// TIA Portal V19 program export: 2 tag tables, 0 data types, 0 data blocks, 1 code blocks (in call order from the OBs), 0 instance data blocks

VAR_GLOBAL   // PLC tag table "Default tag table"
   memstart1 AT %M2.2 : Bool;
END_VAR

VAR_GLOBAL   // PLC tag table "driver"
   "Start Button 0" AT %I0.0 : Bool;
   "Stop Button 0" AT %I0.1 : Bool;
   "Selector 0 (State 0)" AT %I0.2 : Bool;
   "jog left" AT %I0.3 : Bool;
   "jog right" AT %I0.4 : Bool;
   "Potentiometer 0 (V)" AT %IW100 : Int;
   "Belt Conveyor (6m) 0 (V)" AT %QW100 : Int;
   "mem-edge1" AT %M0.0 : Bool;
   "mem-edge2" AT %M0.1 : Bool;
   "mem-edge3" AT %M0.2 : Bool;
   "mem-edge4" AT %M0.3 : Bool;
   "mem-edge5" AT %M0.4 : Bool;
   "memory-start" AT %M1.0 : Bool;
   "memory-stop" AT %M1.1 : Bool;
   "memory-3" AT %M1.2 : Bool;
   "memory-4" AT %M1.3 : Bool;
   "memory-5" AT %M1.4 : Bool;
   "mem-out scale" AT %MD100 : Real;
   "mem-val" AT %MW20 : Int;
   "mem-out norm" AT %MD104 : Real;
   "mem-jog-left" AT %MD108 : Real;
   "mem-jog-right" AT %MD112 : Real;
   spead AT %MD116 : Real;
   spead_enter AT %MD120 : Real;
END_VAR

ORGANIZATION_BLOCK "Main"   // OB1, LAD, ProgramCycle
TITLE = "Main Program Sweep (Cycle)"
{ S7_Optimized_Access := 'TRUE' }
// stored: SetENOAutomatically false
   VAR_INPUT
      Initial_Call : Bool;   // Initial call of this OB
      Remanence : Bool;   // =True, if remanent data are available
   END_VAR
   VAR_TEMP   // added for the SCL form of the ladder/FBD networks
      _w1 : Bool;
      _w2 : Bool;
   END_VAR
BEGIN

REGION Network 1
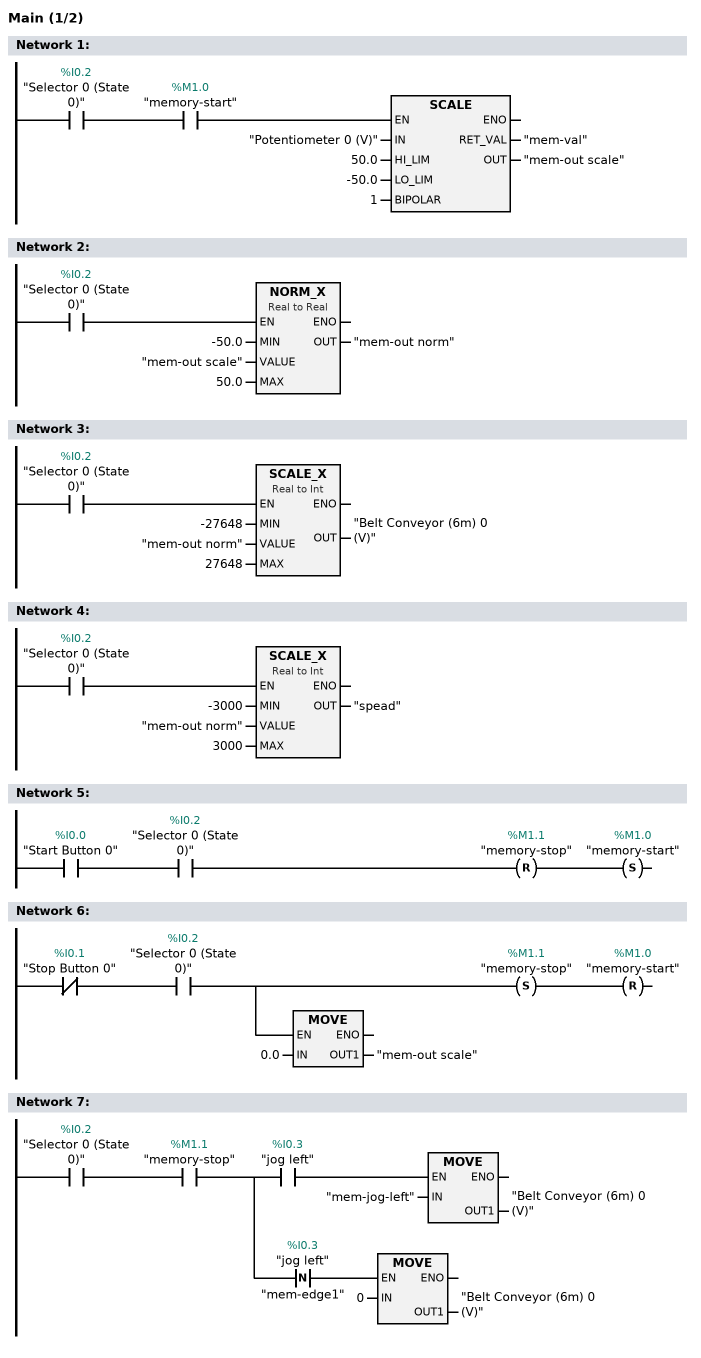
   IF "Selector 0 (State 0)" AND "memory-start" THEN
       "mem-val" := SCALE(IN := "Potentiometer 0 (V)",
                          HI_LIM := 50.0,
                          LO_LIM := -50.0,
                          BIPOLAR := 1,
                          OUT => "mem-out scale");
   END_IF;
END_REGION

REGION Network 2
   RUNG wire#powerrail
      Contact( "Selector 0 (State 0)" )
      { S7_Templates := "[SrcType := Real, DestType := Real]" } Normalize(min := -50.0, value := "mem-out scale", max := 50.0, out => "mem-out norm")
   END_RUNG
   // the same network as SCL:
   IF "Selector 0 (State 0)" THEN
       "mem-out norm" := NORM_X(MIN := -50.0, VALUE := "mem-out scale", MAX := 50.0);
   END_IF;
END_REGION

REGION Network 3
   RUNG wire#powerrail
      Contact( "Selector 0 (State 0)" )
      { S7_Templates := "[SrcType := Real, DestType := Int]" } Scale(min := -27648, value := "mem-out norm", max := 27648, out => "Belt Conveyor (6m) 0 (V)")
   END_RUNG
   // the same network as SCL:
   IF "Selector 0 (State 0)" THEN
       "Belt Conveyor (6m) 0 (V)" := SCALE_X(MIN := -27648, VALUE := "mem-out norm", MAX := 27648);
   END_IF;
END_REGION

REGION Network 4
   RUNG wire#powerrail
      Contact( "Selector 0 (State 0)" )
      { S7_Templates := "[SrcType := Real, DestType := Int]" } Scale(min := -3000, value := "mem-out norm", max := 3000, out => "spead")
   END_RUNG
   // the same network as SCL:
   IF "Selector 0 (State 0)" THEN
       "spead" := SCALE_X(MIN := -3000, VALUE := "mem-out norm", MAX := 3000);
   END_IF;
END_REGION

REGION Network 5
   RUNG wire#powerrail
      Contact( "Start Button 0" )
      Contact( "Selector 0 (State 0)" )
      R_Coil( "memory-stop" )
      S_Coil( "memory-start" )
   END_RUNG
   // the same network as SCL:
   IF "Start Button 0" AND "Selector 0 (State 0)" THEN
       "memory-stop" := FALSE;
       "memory-start" := TRUE;
   END_IF;
END_REGION

REGION Network 6
   RUNG wire#powerrail
      I_Contact( "Stop Button 0" )
      Contact( "Selector 0 (State 0)" )
      wire#w1
      S_Coil( "memory-stop" )
      R_Coil( "memory-start" )
   END_RUNG
   RUNG wire#w1
      Move(in := 0.0, out1 => "mem-out scale")
   END_RUNG
   // the same network as SCL:
   IF NOT "Stop Button 0" AND "Selector 0 (State 0)" THEN
       "memory-stop" := TRUE;
       "memory-start" := FALSE;
       "mem-out scale" := 0.0;
   END_IF;
END_REGION

REGION Network 7
   RUNG wire#powerrail
      Contact( "Selector 0 (State 0)" )
      Contact( "memory-stop" )
      wire#w1
      Contact( "jog left" )
      Move(in := "mem-jog-left", out1 => "Belt Conveyor (6m) 0 (V)")
   END_RUNG
   RUNG wire#w1
      N_Contact(operand := "jog left", bit := "mem-edge1")
      Move(in := 0, out1 => "Belt Conveyor (6m) 0 (V)")
   END_RUNG
   // the same network as SCL:
   #_w1 := "Selector 0 (State 0)" AND "memory-stop";
   IF #_w1 AND "jog left" THEN "Belt Conveyor (6m) 0 (V)" := "mem-jog-left"; END_IF;
   #_w2 := #_w1 AND NOT "jog left" AND "mem-edge1";   // falling edge of "jog left"
   "mem-edge1" := "jog left";
   IF #_w2 THEN "Belt Conveyor (6m) 0 (V)" := 0; END_IF;
END_REGION

REGION Network 8
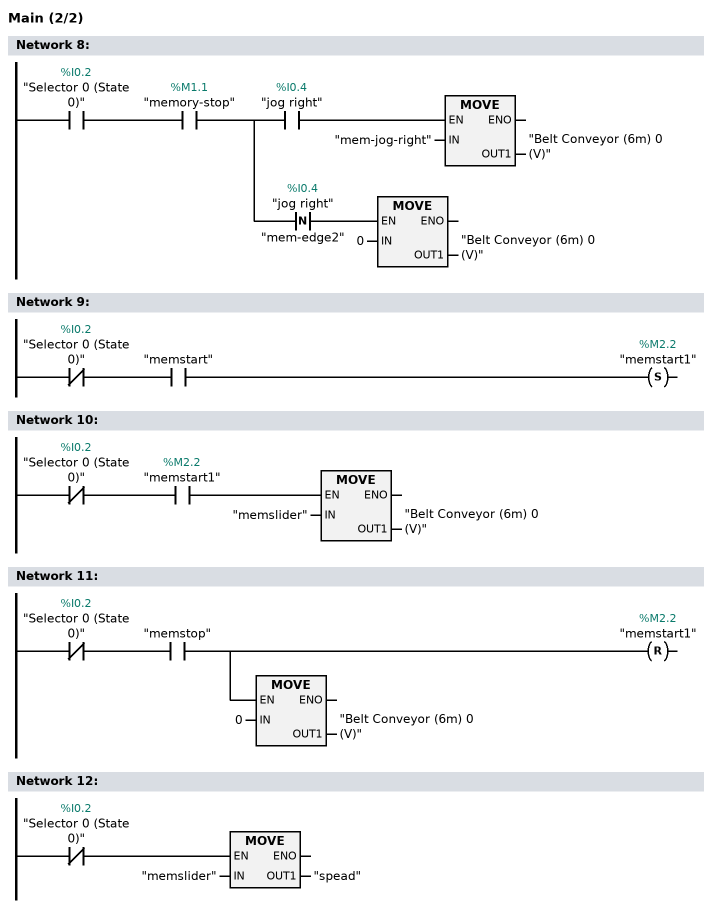
   RUNG wire#powerrail
      Contact( "Selector 0 (State 0)" )
      Contact( "memory-stop" )
      wire#w1
      Contact( "jog right" )
      Move(in := "mem-jog-right", out1 => "Belt Conveyor (6m) 0 (V)")
   END_RUNG
   RUNG wire#w1
      N_Contact(operand := "jog right", bit := "mem-edge2")
      Move(in := 0, out1 => "Belt Conveyor (6m) 0 (V)")
   END_RUNG
   // the same network as SCL:
   #_w1 := "Selector 0 (State 0)" AND "memory-stop";
   IF #_w1 AND "jog right" THEN "Belt Conveyor (6m) 0 (V)" := "mem-jog-right"; END_IF;
   #_w2 := #_w1 AND NOT "jog right" AND "mem-edge2";   // falling edge of "jog right"
   "mem-edge2" := "jog right";
   IF #_w2 THEN "Belt Conveyor (6m) 0 (V)" := 0; END_IF;
END_REGION

REGION Network 9
   RUNG wire#powerrail
      I_Contact( "Selector 0 (State 0)" )
      Contact( "memstart" )
      S_Coil( "memstart1" )
   END_RUNG
   // the same network as SCL:
   IF NOT "Selector 0 (State 0)" AND "memstart" THEN "memstart1" := TRUE; END_IF;
END_REGION

REGION Network 10
   RUNG wire#powerrail
      I_Contact( "Selector 0 (State 0)" )
      Contact( "memstart1" )
      Move(in := "memslider", out1 => "Belt Conveyor (6m) 0 (V)")
   END_RUNG
   // the same network as SCL:
   IF NOT "Selector 0 (State 0)" AND "memstart1" THEN "Belt Conveyor (6m) 0 (V)" := "memslider"; END_IF;
END_REGION

REGION Network 11
   RUNG wire#powerrail
      I_Contact( "Selector 0 (State 0)" )
      Contact( "memstop" )
      wire#w1
      R_Coil( "memstart1" )
   END_RUNG
   RUNG wire#w1
      Move(in := 0, out1 => "Belt Conveyor (6m) 0 (V)")
   END_RUNG
   // the same network as SCL:
   IF NOT "Selector 0 (State 0)" AND "memstop" THEN
       "memstart1" := FALSE;
       "Belt Conveyor (6m) 0 (V)" := 0;
   END_IF;
END_REGION

REGION Network 12
   RUNG wire#powerrail
      I_Contact( "Selector 0 (State 0)" )
      Move(in := "memslider", out1 => "spead")
   END_RUNG
   // the same network as SCL:
   IF NOT "Selector 0 (State 0)" THEN "spead" := "memslider"; END_IF;
END_REGION
END_ORGANIZATION_BLOCK
